// Mitsubishi GX Works2 project: 세탁기능 제어회로   PLC: Q02/Q02H

PROGRAM MAIN
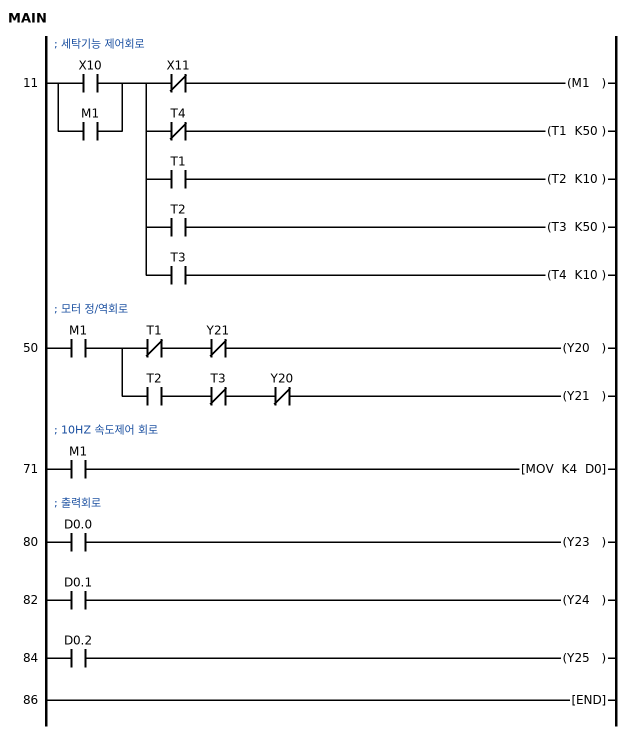
; 세탁기능 제어회로
11    LD      X10
      OR      M1
      MPS
      ANI     X11
      OUT     M1
      MRD
      ANI     T4
      OUT     T1 K50
      MRD
      AND     T1
      OUT     T2 K10
      MRD
      AND     T2
      OUT     T3 K50
      MPP
      AND     T3
      OUT     T4 K10
; 모터 정/역회로
50    LD      M1
      MPS
      ANI     T1
      ANI     Y21
      OUT     Y20
      MPP
      AND     T2
      ANI     T3
      ANI     Y20
      OUT     Y21
; 10HZ 속도제어 회로
71    LD      M1
      MOV     K4 D0
; 출력회로
80    LD      D0.0
      OUT     Y23
82    LD      D0.1
      OUT     Y24
84    LD      D0.2
      OUT     Y25
86    END
END_PROGRAM
